FUNCTION_BLOCK CAC_Average
VAR_INPUT
END_VAR
VAR_OUTPUT
END_VAR
VAR
	Value: REAL;
	Alarm: BOOL;
	OutOfRange: BOOL;
	Offline: BOOL;
END_VAR

VAR_TEMP
	i: INT;
	modbusReal: ModbusUnion;
END_VAR


i:= GVL.nOutputRegisterIndex;
modbusReal.wordValue[1]:= GVL.mb_Output_Registers[i+0];
modbusReal.wordValue[2]:= GVL.mb_Output_Registers[i+1];

Value:= modbusReal.realValue;
GVL.nOutputRegisterIndex:= i+2;


i:= GVL.nOutputCoilIndex;
OutOfRange:= FALSE;
Offline:= GVL.mb_Output_Coils[i+0];
Alarm:= GVL.mb_Output_Coils[i+1];
GVL.nOutputCoilIndex:= i+2;

END_FUNCTION_BLOCK

(* stored: Version 1.1.0.1, ProductVersion 3.1.4024.12
   POU CAC_Average: Id {4795253e-9237-47f6-87a4-7ebf430e31d5}, SpecialFunc None *)
